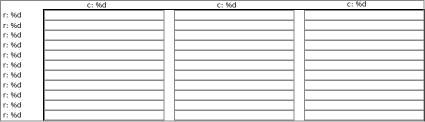
VISUALIZATION _VISU_DefGridTable_raw  // 425x122
VAR_IN_OUT
	mGridTable : ARRAY[0..100, 0..100] OF ST_DeformationPointTbl;
  mGridRowStart : UDINT;
  mGridColStart : UDINT;
END_VAR
    Rectangle (43,9 382x112)
    Frame (44,10 120x10)
        shows _VISU_GridPointView(mGridTable := mGridTable[0+mGridColStart, 0+mGridRowStart])
        pReferences[0]: mGridTable=mGridTable[0+mGridColStart, 0+mGridRowStart]
    Frame (44,20 120x10)
        shows _VISU_GridPointView(mGridTable := mGridTable[0+mGridColStart, 1+mGridRowStart])
        pReferences[0]: mGridTable=mGridTable[0+mGridColStart, 1+mGridRowStart]
    Frame (44,30 120x10)
        shows _VISU_GridPointView(mGridTable := mGridTable[0+mGridColStart, 2+mGridRowStart])
        pReferences[0]: mGridTable=mGridTable[0+mGridColStart, 2+mGridRowStart]
    Frame (44,40 120x10)
        shows _VISU_GridPointView(mGridTable := mGridTable[0+mGridColStart, 3+mGridRowStart])
        pReferences[0]: mGridTable=mGridTable[0+mGridColStart, 3+mGridRowStart]
    Frame (44,50 120x10)
        shows _VISU_GridPointView(mGridTable := mGridTable[0+mGridColStart, 4+mGridRowStart])
        pReferences[0]: mGridTable=mGridTable[0+mGridColStart, 4+mGridRowStart]
    Frame (44,60 120x10)
        shows _VISU_GridPointView(mGridTable := mGridTable[0+mGridColStart, 5+mGridRowStart])
        pReferences[0]: mGridTable=mGridTable[0+mGridColStart, 5+mGridRowStart]
    Frame (44,70 120x10)
        shows _VISU_GridPointView(mGridTable := mGridTable[0+mGridColStart, 6+mGridRowStart])
        pReferences[0]: mGridTable=mGridTable[0+mGridColStart, 6+mGridRowStart]
    Frame (44,80 120x10)
        shows _VISU_GridPointView(mGridTable := mGridTable[0+mGridColStart, 7+mGridRowStart])
        pReferences[0]: mGridTable=mGridTable[0+mGridColStart, 7+mGridRowStart]
    Frame (44,90 120x10)
        shows _VISU_GridPointView(mGridTable := mGridTable[0+mGridColStart, 8+mGridRowStart])
        pReferences[0]: mGridTable=mGridTable[0+mGridColStart, 8+mGridRowStart]
    Frame (44,100 120x10)
        shows _VISU_GridPointView(mGridTable := mGridTable[0+mGridColStart, 9+mGridRowStart])
        pReferences[0]: mGridTable=mGridTable[0+mGridColStart, 9+mGridRowStart]
    Frame (44,110 120x10)
        shows _VISU_GridPointView(mGridTable := mGridTable[0+mGridColStart, 10+mGridRowStart])
        pReferences[0]: mGridTable=mGridTable[0+mGridColStart, 10+mGridRowStart]
    Frame (174,10 120x10)
        shows _VISU_GridPointView(mGridTable := mGridTable[1+mGridColStart, 0+mGridRowStart])
        pReferences[0]: mGridTable=mGridTable[1+mGridColStart, 0+mGridRowStart]
    Frame (174,20 120x10)
        shows _VISU_GridPointView(mGridTable := mGridTable[1+mGridColStart, 1+mGridRowStart])
        pReferences[0]: mGridTable=mGridTable[1+mGridColStart, 1+mGridRowStart]
    Frame (174,30 120x10)
        shows _VISU_GridPointView(mGridTable := mGridTable[1+mGridColStart, 2+mGridRowStart])
        pReferences[0]: mGridTable=mGridTable[1+mGridColStart, 2+mGridRowStart]
    Frame (174,40 120x10)
        shows _VISU_GridPointView(mGridTable := mGridTable[1+mGridColStart, 3+mGridRowStart])
        pReferences[0]: mGridTable=mGridTable[1+mGridColStart, 3+mGridRowStart]
    Frame (174,50 120x10)
        shows _VISU_GridPointView(mGridTable := mGridTable[1+mGridColStart, 4+mGridRowStart])
        pReferences[0]: mGridTable=mGridTable[1+mGridColStart, 4+mGridRowStart]
    Frame (174,60 120x10)
        shows _VISU_GridPointView(mGridTable := mGridTable[1+mGridColStart, 5+mGridRowStart])
        pReferences[0]: mGridTable=mGridTable[1+mGridColStart, 5+mGridRowStart]
    Frame (174,70 120x10)
        shows _VISU_GridPointView(mGridTable := mGridTable[1+mGridColStart, 6+mGridRowStart])
        pReferences[0]: mGridTable=mGridTable[1+mGridColStart, 6+mGridRowStart]
    Frame (174,80 120x10)
        shows _VISU_GridPointView(mGridTable := mGridTable[1+mGridColStart, 7+mGridRowStart])
        pReferences[0]: mGridTable=mGridTable[1+mGridColStart, 7+mGridRowStart]
    Frame (174,90 120x10)
        shows _VISU_GridPointView(mGridTable := mGridTable[1+mGridColStart, 8+mGridRowStart])
        pReferences[0]: mGridTable=mGridTable[1+mGridColStart, 8+mGridRowStart]
    Frame (174,100 120x10)
        shows _VISU_GridPointView(mGridTable := mGridTable[1+mGridColStart, 9+mGridRowStart])
        pReferences[0]: mGridTable=mGridTable[1+mGridColStart, 9+mGridRowStart]
    Frame (174,110 120x10)
        shows _VISU_GridPointView(mGridTable := mGridTable[1+mGridColStart, 10+mGridRowStart])
        pReferences[0]: mGridTable=mGridTable[1+mGridColStart, 10+mGridRowStart]
    Frame (304,10 120x10)
        shows _VISU_GridPointView(mGridTable := mGridTable[2+mGridColStart, 0+mGridRowStart])
        pReferences[0]: mGridTable=mGridTable[2+mGridColStart, 0+mGridRowStart]
    Frame (304,20 120x10)
        shows _VISU_GridPointView(mGridTable := mGridTable[2+mGridColStart, 1+mGridRowStart])
        pReferences[0]: mGridTable=mGridTable[2+mGridColStart, 1+mGridRowStart]
    Frame (304,30 120x10)
        shows _VISU_GridPointView(mGridTable := mGridTable[2+mGridColStart, 2+mGridRowStart])
        pReferences[0]: mGridTable=mGridTable[2+mGridColStart, 2+mGridRowStart]
    Frame (304,40 120x10)
        shows _VISU_GridPointView(mGridTable := mGridTable[2+mGridColStart, 3+mGridRowStart])
        pReferences[0]: mGridTable=mGridTable[2+mGridColStart, 3+mGridRowStart]
    Frame (304,50 120x10)
        shows _VISU_GridPointView(mGridTable := mGridTable[2+mGridColStart, 4+mGridRowStart])
        pReferences[0]: mGridTable=mGridTable[2+mGridColStart, 4+mGridRowStart]
    Frame (304,60 120x10)
        shows _VISU_GridPointView(mGridTable := mGridTable[2+mGridColStart, 5+mGridRowStart])
        pReferences[0]: mGridTable=mGridTable[2+mGridColStart, 5+mGridRowStart]
    Frame (304,70 120x10)
        shows _VISU_GridPointView(mGridTable := mGridTable[2+mGridColStart, 6+mGridRowStart])
        pReferences[0]: mGridTable=mGridTable[2+mGridColStart, 6+mGridRowStart]
    Frame (304,80 120x10)
        shows _VISU_GridPointView(mGridTable := mGridTable[2+mGridColStart, 7+mGridRowStart])
        pReferences[0]: mGridTable=mGridTable[2+mGridColStart, 7+mGridRowStart]
    Frame (304,90 120x10)
        shows _VISU_GridPointView(mGridTable := mGridTable[2+mGridColStart, 8+mGridRowStart])
        pReferences[0]: mGridTable=mGridTable[2+mGridColStart, 8+mGridRowStart]
    Frame (304,100 120x10)
        shows _VISU_GridPointView(mGridTable := mGridTable[2+mGridColStart, 9+mGridRowStart])
        pReferences[0]: mGridTable=mGridTable[2+mGridColStart, 9+mGridRowStart]
    Frame (304,110 120x10)
        shows _VISU_GridPointView(mGridTable := mGridTable[2+mGridColStart, 10+mGridRowStart])
        pReferences[0]: mGridTable=mGridTable[2+mGridColStart, 10+mGridRowStart]
    Rectangle (84,0 40x10), "c: %d", text variable: mGridColStart
    Rectangle (214,0 40x10), "c: %d", text variable: mGridColStart+1
    Rectangle (344,-1 40x10), "c: %d", text variable: mGridColStart+2
    Rectangle (0,10 40x10), "r: %d", text variable: mGridRowStart
    Rectangle (0,20 40x11), "r: %d", text variable: mGridRowStart+1
    Rectangle (0,30 40x10), "r: %d", text variable: mGridRowStart+2
    Rectangle (0,40 40x10), "r: %d", text variable: mGridRowStart+3
    Rectangle (0,50 40x10), "r: %d", text variable: mGridRowStart+4
    Rectangle (0,60 40x10), "r: %d", text variable: mGridRowStart+5
    Rectangle (0,70 40x10), "r: %d", text variable: mGridRowStart+6
    Rectangle (0,80 40x10), "r: %d", text variable: mGridRowStart+7
    Rectangle (0,90 40x10), "r: %d", text variable: mGridRowStart+8
    Rectangle (0,100 40x10), "r: %d", text variable: mGridRowStart+9
    Rectangle (0,110 40x10), "r: %d", text variable: mGridRowStart+10
END_VISUALIZATION

(* stored: Version 1.1.0.1, ProductVersion 3.1.4024.11
   Visu _VISU_DefGridTable_raw: Id {4989c70e-ab93-4913-a9f2-0182b6f94ff4} *)
